// LS Electric XG5000 project: 동남-28
// PLC NewPLC
// module base 0 slot 0: 입출력 모듈:XBC-DN/DP14E (DC 24V 입력 8점, 트랜지스터 출력 6점)

PROGRAM NewProgram (task: 스캔 프로그램)

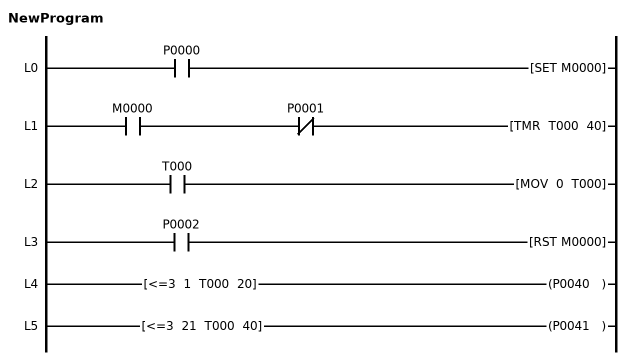
; L0
LOAD      P0000
SET       M0000
; L1
LOAD      M0000
AND NOT   P0001
TMR       T000 40
; L2
LOAD      T000
MOV       0 T000
; L3
LOAD      P0002
RST       M0000
; L4
LOAD<=3   1 T000 20
OUT       P0040
; L5
LOAD<=3   21 T000 40
OUT       P0041